Fanuc KAREL source: ko00005.KL

-- PROVISIONAL review KL for V940-1; original PC SHA256 4292027bf76d9cc2e4422b94319cddc51ad64f9d28a7238746f05a40fed5af73
-- Incomplete behavior may be omitted. Consult companion uncertainty JSON. Do not deploy.
PROGRAM KO00005
%NOLOCKGROUP
-- UNRESOLVED_DECL P1 type=000101
-- UNRESOLVED_DECL P2 type=000101
-- UNRESOLVED_DECL P3 type=000101
-- UNRESOLVED_DECL P4 type=000101
-- UNRESOLVED_DECL OUT type=000101
BEGIN
  -- V9_ZERO_TABLE_METADATA_HINT layout=0001; no indexed target words; source/name/runtime held
  -- UNRESOLVED_PC offsets 5-68; opcodes 27,22,1C,22,1C,22,1C,22,1C,76,7E,4A
  -- UNRESOLVED_PC offsets 73-77; opcodes 7F
END KO00005
